TYPE ST_P3ElectValveName :
STRUCT
		
END_STRUCT
END_TYPE

(* stored: Version 1.1.0.1, ProductVersion 3.1.4024.9
   DUT ST_P3ElectValveName: Id {bf549ee8-c193-47b6-8a1e-4747d910b641} *)
